INTERFACE I_StateModule

PROPERTY CurrentState : UINT
GET
END_GET
END_PROPERTY

END_INTERFACE

(* stored: Version 1.1.0.1, ProductVersion 3.1.4024.12
   Itf I_StateModule: Id {10032349-2530-4511-b9fa-587445f59afa}
   Property CurrentState: Id {9a7bc82b-aa93-4f43-ac51-36077389bf74}
   Get Get: Id {ab125612-6645-4579-acaa-9dcdfbe7bbc3} *)
